// TIA Portal V18 export
ORGANIZATION_BLOCK "Cyclic interrupt"   // OB30, LAD, CyclicInterrupt
{ S7_Optimized_Access := 'TRUE' }
// stored: SetENOAutomatically false
   VAR_INPUT
      Initial_Call : Bool;   // Initial call of this OB
      Event_Count : Int;   // Events discarded
   END_VAR
BEGIN

REGION Network 1
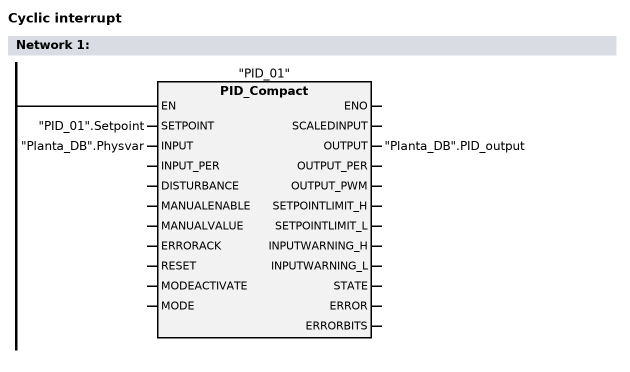
   RUNG wire#powerrail
      "PID_01".PID_Compact(Setpoint := "PID_01".Setpoint, Input := "Planta_DB".Physvar, Input_PER :=, Disturbance :=, ManualEnable :=, ManualValue :=, ErrorAck :=, Reset :=, ModeActivate :=, Mode :=, ScaledInput =>, Output => "Planta_DB".PID_output, Output_PER =>, Output_PWM =>, SetpointLimit_H =>, SetpointLimit_L =>, InputWarning_H =>, InputWarning_L =>, State =>, Error =>, ErrorBits =>)
   END_RUNG
   // the same network as SCL:
   "PID_01"(Setpoint := "PID_01".Setpoint, Input := "Planta_DB".Physvar, Output => "Planta_DB".PID_output);   // PID_Compact
END_REGION
END_ORGANIZATION_BLOCK
